FUNCTION_BLOCK MoveRight EXTENDS GuardMove
VAR_INPUT
END_VAR
VAR_OUTPUT
END_VAR
VAR
END_VAR

(*

short summary
=================
This abstract property returns the class name of the concrete object, 
which is useful for logging/debugging purpose or to check the class name
for ``__DELETE`` in factories (sometimes it's necessary to do more 
than just to free the memory).

.. <legal notes>

legal notes
=================
| SPDX-FileCopyrightText: © 2022 ekvip automation GmbH <info@ekvip.de>
| SPDX-License-Identifier: Apache-2.0
| For details check: Apache-2.0_

.. _Apache-2.0: https://www.apache.org/licenses/LICENSE-2.0

.. </legal notes>

*)
PROPERTY className : CNM_AbstractObject.ClassName
GET
className := 'MoveRight';
END_GET
END_PROPERTY

PROPERTY PROTECTED direction : Rotation
GET
direction := Rotation.RIGHT;
END_GET
END_PROPERTY

END_FUNCTION_BLOCK

(* stored: Version 1.1.0.1
   POU MoveRight: Id {43b7dc69-a2f1-46ab-83de-d917ea897127}, SpecialFunc None
   Property className: Id {68e5fb50-7590-4244-b3e4-8481a248f22b}
   Get Get: Id {f27bef7c-0c22-4d73-a01c-f4c5db9d15fc}
   Property direction: Id {aad34ac8-bebf-4459-827e-66ed4d80b8ce}
   Get Get: Id {a0b760df-b3ec-4bac-87b5-8f8030caf003} *)
